Yaskawa INFORM job: KRIS7.JBI

/JOB
//NAME KRIS7
//POS
///NPOS 337,337,337,19,0,0
///TOOL 0
///POSTYPE PULSE
///PULSE
C00000=36471,-76527,-106813,-19264,71481,-77238
C00001=36471,-76527,-106813,-19264,71481,-77238
C00002=63812,-119516,-80644,27282,71106,-59809
C00003=86670,-29465,-24103,33182,93398,-46515
C00004=88663,-31189,-25266,33292,92471,-45985
C00005=89600,-31952,-25776,33339,92036,-45737
C00006=88663,-31189,-25266,33292,92471,-45985
C00007=88663,-31929,-28188,33361,93666,-45629
C00008=101397,-33118,-34088,22474,91022,-41668
C00009=101397,-32934,-33069,22469,90527,-41762
C00010=101397,-33275,-35023,22483,91481,-41581
C00011=104499,20623,14787,23283,115207,-62973
C00012=104352,17765,12486,23220,115200,-63034
C00013=104529,15851,10717,23303,115245,-62949
C00014=104352,17765,12486,23220,115200,-63034
C00015=100086,19810,13187,22516,115799,-63398
C00016=93288,781,-1160,33549,91987,-44264
C00017=95103,1586,-482,33591,91265,-43744
C00018=95638,1156,-842,33600,91054,-43591
C00019=95103,1586,-482,33591,91265,-43744
C00020=100253,-3614,-11898,25466,91372,-41970
C00021=107199,-8537,-17665,19004,89460,-40114
C00022=108350,-8919,-17473,17740,88760,-39873
C00023=102096,-5783,-13006,25389,90415,-41488
C00024=93175,-13453,-24658,25770,96080,-43586
C00025=29596,-126908,-80456,16683,91164,-67663
C00026=130966,-130992,-81417,-14801,93022,34731
C00027=139735,-123676,-71676,-23223,79574,40827
C00028=138444,-123929,-71735,-23429,79144,40460
C00029=134984,-124514,-71869,-23951,78010,39473
C00030=136755,-124231,-71804,-23689,78586,39979
C00031=136306,-124758,-74432,-23664,79703,39597
C00032=105195,-127447,-79852,-15126,73259,28242
C00033=104798,-126140,-77647,-15190,72530,28198
C00034=108375,-128078,-79564,-15067,73342,29336
C00035=112121,-93277,-65445,-16297,96104,47809
C00036=116095,-84503,-58814,-18813,102506,48434
C00037=114391,-86924,-59797,-19239,101506,47972
C00038=116095,-84503,-58814,-18813,102506,48434
C00039=117812,-129995,-81150,-14641,74986,32390
C00040=118791,-92886,-67151,-14205,85296,31516
C00041=116748,-92781,-67110,-14299,84968,30842
C00042=115499,-92681,-67072,-14351,84774,30431
C00043=116748,-92781,-67110,-14299,84968,30842
C00044=116748,-94243,-70296,-14285,86141,30707
C00045=102870,-92009,-70676,-9222,86435,25689
C00046=102870,-90997,-68303,-9229,85506,25758
C00047=102870,-92009,-70676,-9222,86435,25689
C00048=124106,-98193,-79828,-8318,91183,32632
C00049=120990,-117719,-86799,-1028,78019,-83969
C00050=103618,-122878,-84450,-6731,45671,-69045
C00051=107839,-39273,-43881,-11021,86771,-60654
C00052=104365,-32496,-38210,-6982,87775,-60806
C00053=106442,-32422,-37791,-10039,91664,-60187
C00054=103260,-36857,-40680,-8847,97536,-61636
C00055=110992,-39766,-43585,-17340,97602,-59383
C00056=111851,-103912,-94699,-10334,87868,-68255
C00057=100525,-93554,-87313,-9422,87254,-72087
C00058=95765,-72558,-76889,-7644,100510,-59309
C00059=95463,-76426,-71939,-16938,115118,-61391
C00060=97889,-71418,-68275,-18856,117864,-61016
C00061=108072,-63754,-61449,-27079,123073,-58329
C00062=126453,-110744,-88068,-25157,96958,-85114
C00063=124515,-113648,-86106,-25282,93913,-85187
C00064=121942,-111698,-85261,-25663,93564,-86071
C00065=117176,-108078,-83892,-26284,92993,-87738
C00066=122754,-106725,-87203,-25770,97209,-86568
C00067=142865,-91008,-85242,-17891,113758,-73123
C00068=142005,-90205,-84914,-18160,113770,-73464
C00069=93871,-48257,-54590,14207,101968,48555
C00070=106716,17042,-5346,15024,102835,53222
C00071=114740,-14345,-34597,13608,101053,59815
C00072=127078,-3386,-21930,8482,103399,53955
C00073=129218,-1885,-18027,7623,102641,53139
C00074=128838,-13728,-23209,15330,113259,56406
C00075=127376,-6452,-15191,17883,117233,55977
C00076=122058,-3228,-13278,23261,119236,52777
C00077=102997,28917,14853,20600,116287,84527
C00078=102837,-6052,-12869,23266,105489,87265
C00079=105472,-3409,-10021,23525,105335,88236
C00080=105487,-912,-7016,26090,105184,88300
C00081=104416,1445,-8009,23523,106791,88129
C00082=100743,5943,-9423,11985,113108,51981
C00083=104100,-22795,-28366,25068,61310,50210
C00084=122112,-33809,-21710,17217,45375,58941
C00085=131285,-32631,-21327,509,47900,55790
C00086=127059,-25073,-15738,7623,47605,53752
C00087=124156,-6831,-1542,11317,48078,52428
C00088=117469,-7945,-6130,22808,51414,49873
C00089=27812,-119319,-87277,42007,83182,24370
C00090=5621,-139291,-109992,39952,96377,-80222
C00091=5621,-139291,-109992,39952,96377,-80222
C00092=2821,-156918,-126127,-8650,50468,-54614
C00093=2821,-156918,-126127,-8650,75949,-54614
C00094=-114520,-110749,-78127,-8650,75949,-54614
C00095=-130701,-93848,-55732,21077,70446,-8081
C00096=-119736,-94913,-51299,8905,54174,-4125
C00097=-119736,-93106,-48364,9003,53306,-4201
C00098=-119736,-91977,-46540,9068,52768,-4251
C00099=-119736,-92203,-46902,9053,52876,-4241
C00100=-119787,-88445,-45584,8939,53987,-4163
C00101=-119736,-93071,-48307,9005,53289,-4204
C00102=-119736,-93071,-48307,9005,53289,-4204
C00103=-119736,-93071,-48307,9005,53289,-4204
C00104=-119736,-92181,-46869,9053,52867,-4244
C00105=-119736,-92317,-47089,9045,52931,-4239
C00106=-119771,-89498,-46107,8960,53770,-4179
C00107=-119736,-93267,-48625,8993,53383,-4198
C00108=-119736,-93267,-48625,8993,53383,-4198
C00109=-119736,-93267,-48625,8993,53383,-4198
C00110=-119736,-92320,-47093,9047,52931,-4240
C00111=-119736,-92484,-47359,9038,53009,-4233
C00112=-119776,-89491,-46317,8947,53899,-4170
C00113=-119736,-93550,-49086,8979,53518,-4188
C00114=-119736,-95350,-52013,8882,54384,-4113
C00115=-114361,-95392,-52404,-9141,55279,249
C00116=-114361,-93732,-49694,-9231,54474,321
C00117=-114361,-92426,-47572,-9302,53848,379
C00118=-114361,-92561,-47791,-9294,53912,373
C00119=-114623,-89431,-46697,-9121,54806,189
C00120=-114361,-93574,-49437,-9237,54399,330
C00121=-157280,-84649,-46195,2979,55353,-16615
C00122=-157280,-84384,-45724,2984,55199,-16619
C00123=-157280,-83620,-44370,2999,54759,-16630
C00124=-157280,-83726,-44557,2996,54820,-16629
C00125=-155888,-80713,-43363,2571,55586,-16063
C00126=-157843,-85963,-46912,3146,55137,-16842
C00127=-186482,-48100,-18697,2331,50903,-27233
C00128=-187472,-46614,-16803,2745,50531,-27658
C00129=-187472,-45763,-15021,2772,49872,-27676
C00130=-187472,-45864,-15234,2769,49950,-27673
C00131=-185259,-43079,-13610,1852,50319,-26729
C00132=-186728,-50494,-20137,2443,50566,-27343
C00133=-173177,-79635,-34784,14301,47494,-39802
C00134=-170114,-73061,-28660,13270,46626,-38584
C00135=-119904,-88221,-34141,-8998,40682,-15980
C00136=-119767,-102866,-45459,-9162,40143,-15856
C00137=-114881,-103501,-45094,-2719,38974,-10407
C00138=-106437,-88415,-33714,-6684,40170,-6473
C00139=-59844,-64383,-24187,-21266,54434,11788
C00140=-55872,-59424,-21793,-21840,56429,13005
C00141=-56728,-59811,-20829,-16196,48671,13044
C00142=-60192,-86606,-39094,-15561,45595,12032
C00143=-156319,-84382,-37772,-22252,46282,-6119
C00144=-155863,-75602,-29197,-22688,45688,-5754
C00145=-171147,-77982,-28397,2458,37476,-29192
C00146=-189524,-53452,-17206,6300,43588,-32690
C00147=-192814,-47813,-14131,7829,44864,-34109
C00148=-192943,-40170,-9756,2318,45440,-29171
C00149=-168938,-74165,-32389,-22140,45247,-8707
C00150=-139665,-98627,-47692,-8234,50597,-7190
C00151=-157202,-83214,-35232,9186,49733,-29053
C00152=-99055,-87999,-36568,-9269,48061,-5453
C00153=-70072,-109159,-59979,-19142,60032,12699
C00154=-153403,-114623,-61310,-4271,48117,-12926
C00155=-150942,-88287,-33092,-1923,37824,-12225
C00156=-192456,-54522,-18938,15787,50129,-30195
C00157=-191005,-51820,-17697,10248,48517,-24206
C00158=-191538,-49735,-14965,7448,44104,-24349
C00159=-196130,-40875,-10027,9488,46067,-26268
C00160=-193358,-74104,-32741,8607,42709,-25326
C00161=-183204,-85382,-41090,22318,63247,-34683
C00162=-169612,-75107,-30908,21185,58925,-30299
C00163=-165096,-78115,-32117,20755,57090,-28885
C00164=-103759,-88277,-35558,4643,44290,-5139
C00165=-64684,-68765,-27814,-9350,50752,11304
C00166=-59734,-63411,-25340,-10717,52547,13159
C00167=-53928,-55634,-21454,-12166,54909,15247
C00168=-72635,-96956,-47079,-7004,47380,8249
C00169=2821,-156918,-126127,-8650,75949,-54614
C00170=2821,-156918,-126127,-8650,50468,-54614
C00171=5621,-139291,-109992,39952,96377,-80222
C00172=5621,-139291,-109992,39952,96377,-80222
C00173=5621,-139291,-109992,39952,96377,-80222
C00174=5621,-139291,-109992,39952,96377,-80222
C00175=2821,-156918,-126127,-8650,50468,-54614
C00176=2821,-156918,-126127,-8650,75949,-54614
C00177=-103466,-143035,-89833,-18127,44217,664
C00178=-153034,-42791,-3789,574,51224,-21077
C00179=-154411,-23786,22188,-6392,45845,-11810
C00180=-163692,-14831,30793,-3045,43978,-15753
C00181=-162658,-12144,32796,-3380,44162,-15317
C00182=-162658,-10372,35929,-3443,43146,-15280
C00183=-162658,-10822,35136,-3427,43403,-15291
C00184=-163644,-13399,33193,-3102,43239,-15709
C00185=-163644,-12612,34572,-3127,42795,-15690
C00186=-163043,-11060,35746,-3327,42891,-15434
C00187=-163515,-12286,34819,-3170,42815,-15635
C00188=-166152,-32133,5550,-1997,50546,-16952
C00189=-100006,-46830,-3879,-17345,57754,8477
C00190=-55652,-4276,24712,-7053,56203,22524
C00191=-58398,37345,76759,-13956,42466,23962
C00192=-66063,-5406,39790,-11450,41903,20618
C00193=-66063,-3286,43507,-11723,40729,20781
C00194=-66063,-4032,42206,-11625,41137,20723
C00195=-64962,-6235,40444,-12035,41233,21210
C00196=-64962,-5161,42315,-12179,40646,21295
C00197=-65448,-4202,43083,-11996,40600,21078
C00198=-65121,-4851,42561,-12118,40631,21223
C00199=-65121,-17453,19695,-10602,48085,20268
C00200=-72607,-39142,3670,-8250,46011,17274
C00201=-104110,-83683,-24495,4068,39615,3407
C00202=-151806,-110432,-47458,34093,62536,-28079
C00203=-114089,-66317,-11235,33609,49333,-16712
C00204=-80530,-20506,23368,24271,40665,-3524
C00205=-74745,-11317,36142,23442,36289,-1903
C00206=-74745,-9368,39521,24041,35298,-2233
C00207=-85567,-6911,52266,59999,33710,-18160
C00208=-84359,-5993,52985,59939,33118,-17833
C00209=-75543,-10512,38192,25890,35469,-3179
C00210=-78021,-4049,43264,26836,36333,-4217
C00211=-78021,-4049,43264,26836,36333,-4217
C00212=-78560,-2493,44527,27046,36504,-4446
C00213=-78021,-4049,43264,26836,36333,-4217
C00214=-84671,-29838,2091,23749,49176,-3555
C00215=-92002,99,24477,25497,52744,-5935
C00216=-90066,7053,36780,26343,48553,-6224
C00217=-86465,14687,47675,26361,44982,-5590
C00218=-86465,16658,51362,26930,43852,-5949
C00219=-92154,15823,55176,43758,42694,-12452
C00220=-91010,16935,56226,43590,42132,-12113
C00221=-87466,14565,48542,29200,44405,-6685
C00222=-88476,20167,53834,29701,44402,-7193
C00223=-88765,21892,55502,29860,44374,-7348
C00224=-89073,23808,57378,30039,44325,-7522
C00225=-88765,21892,55502,29860,44374,-7348
C00226=-92823,2508,20138,26462,56153,-5606
C00227=-93465,20990,41911,27889,52866,-6816
C00228=-91045,28828,52484,28118,49890,-6598
C00229=-91045,30451,55705,28580,48873,-6919
C00230=-95613,30623,60677,42443,47375,-11939
C00231=-94901,31380,61454,42363,46989,-11750
C00232=-91803,28745,53220,30282,49450,-7369
C00233=-95909,-7710,13963,29350,55596,-7301
C00234=-94576,-67258,-23025,-57506,77870,531
C00235=-146401,-54758,-1647,-68188,44391,-5039
C00236=-142614,-8623,29205,-63903,48682,-7044
C00237=-144464,20682,60858,-67736,45663,-4895
C00238=-144464,22107,63347,-68464,45346,-4423
C00239=-144027,21529,62623,-69515,45942,-4175
C00240=-144859,22233,63313,-69675,45420,-4267
C00241=-144060,21537,62613,-69510,45926,-4186
C00242=-141431,-828,33685,-64125,50152,-7263
C00243=-141985,-10259,26135,-64166,52154,-6525
C00244=-141985,6399,55921,-71703,48228,-1192
C00245=-146205,13772,66109,-74932,44993,-221
C00246=-146205,16430,70459,-76214,44629,596
C00247=-146205,13772,66109,-74932,44993,-221
C00248=-147267,14605,66894,-75256,44365,-306
C00249=-146205,13772,66109,-74932,44993,-221
C00250=-145528,19198,71305,-75151,45267,107
C00251=-145166,21952,74026,-75304,45401,306
C00252=-144772,25167,77279,-75529,45528,563
C00253=-145166,21952,74026,-75304,45401,306
C00254=-145571,-16681,30939,-69324,47370,-3717
C00255=-149532,-31410,21037,-71230,44475,-3428
C00256=-151069,-17310,48414,-81811,41046,2644
C00257=-155207,-6338,62509,-87203,38392,4585
C00258=-155206,-3775,66483,-88647,38310,5410
C00259=-155207,-6338,62509,-87203,38392,4585
C00260=-156672,-5360,63276,-87839,37607,4518
C00261=-155207,-6338,62509,-87203,38392,4585
C00262=-153924,-2552,65524,-86505,39089,4564
C00263=-153389,-833,66935,-86244,39378,4573
C00264=-152779,1247,68674,-85973,39703,4598
C00265=-153389,-833,66935,-86244,39378,4573
C00266=-127211,-52277,-10135,-62715,61377,-4297
C00267=-127211,-63632,-31775,-59501,65152,-7618
C00268=-137468,-45448,-13164,-23993,62707,-9546
C00269=-142031,-34381,-3630,-18745,59946,-9254
C00270=-153480,-23481,18954,-7895,48240,-10284
C00271=-154837,-15674,32352,-7510,43874,-10435
C00272=-154881,-15642,32376,-7496,43872,-10454
C00273=-163905,-10778,37737,-6230,39530,-12164
C00274=-163679,-4139,45223,-21101,38086,-2029
C00275=-164728,-2193,48881,-26376,35092,-528
C00276=-146970,-27557,19782,-29282,44621,5055
C00277=-77984,-28544,12598,-9594,52255,4511
C00278=-87329,-14910,33502,8192,43267,-2149
C00279=-87274,-14870,33531,8174,43265,-2126
C00280=-77526,-7325,39164,4963,42972,2054
C00281=-74703,-2158,47540,17953,35749,-596
C00282=-74957,-595,50445,22566,33903,-2166
C00283=-84696,-19604,28451,27180,39406,-6073
C00284=-87454,-109874,-47340,27972,40441,-7116
C00285=-87454,-109874,-47340,27972,40441,-7116
C00286=-82765,-14870,18327,18756,64283,-30139
C00287=-70453,-8973,33300,17854,53830,-23621
C00288=-79133,18874,57440,18465,54102,-25119
C00289=-78473,16959,55330,17021,52555,-21596
C00290=-81801,-8338,17757,15293,62207,-20035
C00291=-80465,5283,36828,18721,53635,-17767
C00292=-81257,8258,39312,19057,54012,-18385
C00293=-86289,31654,62323,20130,49904,-23761
C00294=-86244,31688,62797,19436,47278,-24020
C00295=-89829,15295,36039,20471,54300,-28399
C00296=-88516,27412,50085,20716,51710,-28378
C00297=-88101,27329,53482,18902,40394,-29830
C00298=-85023,22588,57884,12283,20397,-30375
C00299=-84309,12450,52732,13133,12354,-31131
C00300=-84341,-54767,463,16268,10060,-32559
C00301=-89075,-25175,21935,52893,15017,-40843
C00302=-80632,-262,47578,28811,6370,-27546
C00303=-80188,4143,51700,27800,5999,-27018
C00304=-78793,13633,71285,-46780,-2668,6342
C00305=-83238,-13210,39391,48775,6583,-36846
///LIMIT ON
C00306=-68361,-31604,26984,-58103,4691,13513
///LIMIT OFF
C00307=-66564,-14119,49098,-114271,5370,38931
C00308=-64215,-1164,72142,-148990,11349,55050
///LIMIT ON
C00309=-70339,-38157,28491,-125542,3279,43165
///LIMIT OFF
C00310=-80839,-71335,-37546,-3712,65478,-21646
C00311=-155891,-91755,-42787,-14200,56541,28985
C00312=-171260,-20220,18318,-13706,55116,27713
C00313=-175592,-12005,31520,-10745,48833,21454
C00314=-167202,11927,51151,-10059,48724,20347
C00315=-164608,7730,50211,-16502,43624,19417
C00316=-166381,-4712,22713,-7153,56786,16501
C00317=-164906,4240,35250,-11113,52340,17926
C00318=-163520,9172,39392,-11480,52509,18470
C00319=-157524,37432,66627,-13367,51178,21072
C00320=-157651,33997,63941,-13772,48810,17620
C00321=-157953,21876,39059,-9901,58764,16683
C00322=-154411,30422,52036,-17366,53831,19464
C00323=-154093,33138,54821,-17521,53595,19641
C00324=-155920,26750,56620,-12911,32167,21130
C00325=-156729,27540,61020,-9631,24538,20676
C00326=-159295,5897,40777,-3469,23124,17976
C00327=-161800,-2337,33413,-1605,23382,16874
C00328=-162218,5196,42221,-1134,21829,16584
C00329=-163744,11950,58915,1437,15023,15129
C00330=-178555,-20714,28140,24908,19354,1618
C00331=-170517,-15099,37122,-3989,15402,13548
C00332=-166794,-3567,48220,-19541,26132,18647
C00333=-176772,-46405,12054,26858,15885,1020
C00334=-187852,-124872,-80037,-26712,55091,17871
C00335=-130728,-161100,-136081,-16173,33339,28558
C00336=-1271,-161100,-136081,-16173,33339,28558
BC00000=295309,515546,1075134
BC00001=295309,515546,1075134
BC00002=396955,458142,797628
BC00003=396955,458142,797628
BC00004=396955,458142,797628
BC00005=396955,458142,797628
BC00006=396955,458142,797628
BC00007=396955,458142,797628
BC00008=396955,458142,797628
BC00009=396955,458142,797628
BC00010=396955,458142,797628
BC00011=396955,458142,797628
BC00012=396955,458142,797628
BC00013=396955,458142,797628
BC00014=396955,458142,797628
BC00015=396955,458142,797628
BC00016=396955,458142,797628
BC00017=396955,458142,797628
BC00018=396955,458142,797628
BC00019=396955,458142,797628
BC00020=396955,458142,797628
BC00021=396955,458142,797628
BC00022=396955,458142,797628
BC00023=396955,458142,797628
BC00024=396955,458142,797628
BC00025=396955,458142,797628
BC00026=1315,458142,797628
BC00027=1315,355292,797628
BC00028=1315,355292,797628
BC00029=1315,355292,797628
BC00030=1315,355292,797628
BC00031=1315,355292,797628
BC00032=1315,355292,797628
BC00033=1315,355292,797628
BC00034=1315,355292,797628
BC00035=1315,355292,797628
BC00036=1315,355292,797628
BC00037=1315,355292,797628
BC00038=1315,355292,797628
BC00039=1315,355292,797628
BC00040=1315,355292,797628
BC00041=1315,355292,797628
BC00042=1315,355292,797628
BC00043=1315,355292,797628
BC00044=1315,355292,797628
BC00045=1315,355292,797628
BC00046=1315,355292,797628
BC00047=1315,355292,797628
BC00048=1315,355292,797628
BC00049=1056,429044,516729
BC00050=1056,362244,516729
BC00051=1055,360438,517007
BC00052=786,360252,517036
BC00053=1003,360221,517041
BC00054=1055,360214,517042
BC00055=1055,360214,517042
BC00056=752,360214,695044
BC00057=752,360214,695044
BC00058=752,360214,695044
BC00059=752,360214,695044
BC00060=752,360214,695044
BC00061=752,360214,695044
BC00062=752,360214,695044
BC00063=752,360214,695044
BC00064=752,360214,695044
BC00065=752,360214,695044
BC00066=752,360214,695044
BC00067=752,360214,695044
BC00068=752,503342,695044
BC00069=396955,508258,797628
BC00070=396955,458142,797628
BC00071=396955,458142,797628
BC00072=396955,458142,797628
BC00073=396955,458142,797628
BC00074=396955,458142,797628
BC00075=396955,458142,797628
BC00076=396955,458142,797628
BC00077=396955,458142,797628
BC00078=396955,458142,797628
BC00079=396955,458142,797628
BC00080=396955,458142,797628
BC00081=396955,458142,797628
BC00082=396955,458142,797628
BC00083=396955,458142,516729
BC00084=396955,458142,516729
BC00085=396955,458142,516729
BC00086=396956,458130,516729
BC00087=396955,458142,516729
BC00088=396955,458142,516729
BC00089=396955,458142,516729
BC00090=188270,458142,1013387
BC00091=188270,415623,1052769
BC00092=159481,115072,1070630
BC00093=159481,2193,1070630
BC00094=222221,2193,888573
BC00095=343723,4817,818861
BC00096=343723,4817,818861
BC00097=343723,4817,818861
BC00098=343723,4817,818861
BC00099=343723,4817,818861
BC00100=343723,4817,818861
BC00101=343723,4817,818861
BC00102=285503,4817,818861
BC00103=285503,5201,817244
BC00104=285503,5201,817244
BC00105=285503,5201,817244
BC00106=285503,5201,817244
BC00107=285503,5201,817244
BC00108=225351,5201,824692
BC00109=225351,5201,816215
BC00110=225351,5201,816215
BC00111=225351,5201,816215
BC00112=225351,5201,816215
BC00113=225351,5201,816215
BC00114=225351,5201,816215
BC00115=193660,5201,816215
BC00116=193660,5201,816215
BC00117=193660,5201,816215
BC00118=193660,5201,816215
BC00119=193660,5201,816215
BC00120=193660,5201,816215
BC00121=193660,5201,816215
BC00122=193660,5201,816215
BC00123=193660,5201,816215
BC00124=193660,5201,816215
BC00125=193660,5201,816215
BC00126=193660,5201,816215
BC00127=207415,5201,867665
BC00128=207415,5201,867665
BC00129=207415,5201,867665
BC00130=207415,5201,867665
BC00131=207415,5201,867665
BC00132=207415,5201,867665
BC00133=207415,5201,867665
BC00134=207415,5201,867665
BC00135=207415,5201,867665
BC00136=207415,5201,867665
BC00137=273654,5201,867665
BC00138=273654,5201,867665
BC00139=273654,5201,867665
BC00140=273654,5201,867665
BC00141=273654,5201,867665
BC00142=273654,5201,867665
BC00143=273654,5201,867665
BC00144=225140,12373,867665
BC00145=225140,12373,867665
BC00146=206995,12373,867665
BC00147=206995,12373,867665
BC00148=206995,12373,867665
BC00149=206995,12373,867665
BC00150=268142,12373,867665
BC00151=268142,12373,867665
BC00152=268142,12373,867665
BC00153=268142,12373,867665
BC00154=254581,12373,867665
BC00155=254581,12373,867665
BC00156=254581,12373,867665
BC00157=206517,12373,867665
BC00158=206517,12373,867665
BC00159=206517,12373,867665
BC00160=206517,12373,867665
BC00161=267255,12373,867665
BC00162=267255,12373,867665
BC00163=267255,12373,867665
BC00164=267255,12373,867665
BC00165=267255,12373,867665
BC00166=267255,12373,867665
BC00167=267255,12373,867665
BC00168=267255,12373,867665
BC00169=159481,2193,1070630
BC00170=159481,115072,1070630
BC00171=188270,458142,1013387
BC00172=188270,529869,1013387
BC00173=188270,458142,1013387
BC00174=188270,415623,1052769
BC00175=159481,115072,1070630
BC00176=159481,2193,1070630
BC00177=256379,66753,1051189
BC00178=187914,126248,1051189
BC00179=187914,126248,1051189
BC00180=187915,126247,1051163
BC00181=187915,126247,1051163
BC00182=187915,126247,1051163
BC00183=187915,126247,1051163
BC00184=187915,126247,1051163
BC00185=187915,126247,1051163
BC00186=187915,126247,1051163
BC00187=187915,126247,1051163
BC00188=187915,126247,1051163
BC00189=237533,126248,1051189
BC00190=187914,126248,1051189
BC00191=187914,99975,1051189
BC00192=235697,126248,1051189
BC00193=235697,126248,1051189
BC00194=235697,126248,1051189
BC00195=235697,126248,1051189
BC00196=235697,126248,1051189
BC00197=235697,126248,1051189
BC00198=235697,126248,1051189
BC00199=235697,126248,1051189
BC00200=235697,126248,1051189
BC00201=235697,126248,1051189
BC00202=291851,64960,1051189
BC00203=291851,64960,1051189
BC00204=244068,34238,1051189
BC00205=244068,34238,1051189
BC00206=244068,34238,1051189
BC00207=244068,34238,1051189
BC00208=244068,34238,1051189
BC00209=244068,34238,1051189
BC00210=244068,34238,1051189
BC00211=244068,34238,1051189
BC00212=244068,34238,1051189
BC00213=244068,34238,1051189
BC00214=244068,34238,1051189
BC00215=244068,34238,1051189
BC00216=244068,34238,1051189
BC00217=244068,34238,1051189
BC00218=244068,34238,1051189
BC00219=244068,34238,1051189
BC00220=244068,34238,1051189
BC00221=244068,34238,1051189
BC00222=244068,34238,1051189
BC00223=244068,34238,1051189
BC00224=244068,34238,1051189
BC00225=244068,34238,1051189
BC00226=244068,34238,1051189
BC00227=244068,34238,1051189
BC00228=244067,34238,1051186
BC00229=244067,34238,1051186
BC00230=244067,34238,1051186
BC00231=244067,34238,1051186
BC00232=244067,34238,1051186
BC00233=244067,34238,1051186
BC00234=244067,64961,1051183
BC00235=198013,64961,1051183
BC00236=198013,64961,1051183
BC00237=198013,47917,1051183
BC00238=198013,47917,1051183
BC00239=198013,47917,1051183
BC00240=198013,47917,1051183
BC00241=198013,47917,1051183
BC00242=198013,47917,1051183
BC00243=198013,47917,1051183
BC00244=198013,47917,1051183
BC00245=198013,47917,1051183
BC00246=198013,47917,1051183
BC00247=198013,47917,1051183
BC00248=198013,47917,1051183
BC00249=198013,47917,1051183
BC00250=198013,47917,1051183
BC00251=198013,47917,1051183
BC00252=198013,47917,1051183
BC00253=198013,47917,1051183
BC00254=198013,47917,1051183
BC00255=198013,47917,1051183
BC00256=198013,47917,1051183
BC00257=198013,47917,1051183
BC00258=198013,47917,1051183
BC00259=198013,47917,1051183
BC00260=198013,47917,1051183
BC00261=198013,47917,1051183
BC00262=198013,47917,1051183
BC00263=198013,47917,1051183
BC00264=198013,47917,1051183
BC00265=198013,47917,1051183
BC00266=198013,47917,1051183
BC00267=198013,47917,1051183
BC00268=180161,98336,1051187
BC00269=182927,108294,1051188
BC00270=187693,125451,1051189
BC00271=187914,126248,1051189
BC00272=187914,126248,1051189
BC00273=187914,126248,1051189
BC00274=187914,126248,1051189
BC00275=187914,126248,1051189
BC00276=187914,126248,1051189
BC00277=244068,126248,1051189
BC00278=244068,126248,1051189
BC00279=244068,126248,1051189
BC00280=244068,126248,1051189
BC00281=244068,126248,1051189
BC00282=244068,126248,1051189
BC00283=244068,126248,1051189
BC00284=244068,126248,1051189
BC00285=244068,64960,1051189
BC00286=244068,34238,1051189
BC00287=244068,34238,1051189
BC00288=244068,34238,1051189
BC00289=244068,34238,1051189
BC00290=244068,34238,1051189
BC00291=244068,34238,1051189
BC00292=244068,34238,1051189
BC00293=244068,34238,1051189
BC00294=244068,34238,1051189
BC00295=244068,34238,1051189
BC00296=244068,34238,1051189
BC00297=244068,34238,1051189
BC00298=244068,34238,1051189
BC00299=244068,34238,1051189
BC00300=244068,64960,1051189
BC00301=244068,34238,1051189
BC00302=244068,34238,1051189
BC00303=244068,34238,1051186
BC00304=244068,34238,1051189
BC00305=244068,34238,1051189
BC00306=244068,34238,1051189
BC00307=244067,34238,1051187
BC00308=244068,34238,1051189
BC00309=244068,34238,1051189
BC00310=244068,34238,1051189
BC00311=193074,64960,1051189
BC00312=193074,32459,1055846
BC00313=193074,32459,1055846
BC00314=193074,32459,1055846
BC00315=193075,32459,1055844
BC00316=193074,32459,1055846
BC00317=193074,32459,1055846
BC00318=193074,32459,1055846
BC00319=193074,32459,1055846
BC00320=193074,32459,1055846
BC00321=193074,32459,1055846
BC00322=193074,32459,1055846
BC00323=193074,32459,1055846
BC00324=193074,32459,1055845
BC00325=193074,32459,1055846
BC00326=193074,32459,1055846
BC00327=193074,32459,1055846
BC00328=193074,32459,1055846
BC00329=193074,32459,1055846
BC00330=211313,32459,1055846
BC00331=193074,32459,1055846
BC00332=193074,32459,1055846
BC00333=193074,32459,1055846
BC00334=292209,32459,1055846
BC00335=189350,71534,1070791
BC00336=189350,455301,1070791
EC00000=0,-183832
EC00001=88685,372644
EC00002=88685,372644
EC00003=88685,372644
EC00004=88685,372644
EC00005=88685,372644
EC00006=88685,372644
EC00007=88685,372644
EC00008=88685,372644
EC00009=88685,372644
EC00010=88685,372644
EC00011=88685,372644
EC00012=88685,372644
EC00013=88685,372644
EC00014=88685,372644
EC00015=88685,372644
EC00016=88685,372644
EC00017=88685,372644
EC00018=88685,372644
EC00019=88685,372644
EC00020=88685,372644
EC00021=88685,372644
EC00022=88685,372644
EC00023=88685,372644
EC00024=88685,372644
EC00025=88685,372644
EC00026=88685,372644
EC00027=88685,372644
EC00028=88685,372644
EC00029=88685,372644
EC00030=88685,372644
EC00031=88685,372644
EC00032=88685,372644
EC00033=88685,372644
EC00034=88685,372644
EC00035=88685,372644
EC00036=88685,372644
EC00037=88685,372644
EC00038=88685,372644
EC00039=88685,372644
EC00040=88685,372644
EC00041=88685,372644
EC00042=88685,372644
EC00043=88685,372644
EC00044=88685,372644
EC00045=88685,372644
EC00046=88685,372644
EC00047=88685,372644
EC00048=88685,372644
EC00049=-264893,372644
EC00050=-264893,372644
EC00051=-264346,372644
EC00052=-264290,372644
EC00053=-264280,372644
EC00054=-264278,372644
EC00055=-264278,372644
EC00056=85879,372644
EC00057=85879,372644
EC00058=85879,372644
EC00059=85879,372644
EC00060=85879,372644
EC00061=85879,372644
EC00062=85879,372644
EC00063=85879,372644
EC00064=85879,372644
EC00065=85879,372644
EC00066=85879,372644
EC00067=85879,372644
EC00068=85879,372644
EC00069=88685,372644
EC00070=88685,372644
EC00071=88685,428210
EC00072=88685,428210
EC00073=88685,428210
EC00074=88685,428210
EC00075=88685,428210
EC00076=88685,428210
EC00077=88685,372644
EC00078=88685,372644
EC00079=88685,372644
EC00080=88685,372644
EC00081=88685,372644
EC00082=88685,372644
EC00083=-264893,372644
EC00084=-264893,421244
EC00085=-264893,421244
EC00086=-264894,421244
EC00087=-264893,421244
EC00088=-264893,421244
EC00089=-264893,372644
EC00090=-264890,372644
EC00091=-264890,372644
EC00092=196570,372645
EC00093=492199,372645
EC00094=492199,372645
EC00095=492199,372645
EC00096=492199,372645
EC00097=492199,372645
EC00098=492199,372645
EC00099=492199,372645
EC00100=492199,372645
EC00101=492199,372645
EC00102=492199,372645
EC00103=492199,372645
EC00104=492199,372645
EC00105=492199,372645
EC00106=492199,372645
EC00107=492199,372645
EC00108=492199,372645
EC00109=492199,372645
EC00110=492199,372645
EC00111=492199,372645
EC00112=492199,372645
EC00113=492199,372645
EC00114=492199,372645
EC00115=492199,372645
EC00116=492199,372645
EC00117=492199,372645
EC00118=492199,372645
EC00119=492199,372645
EC00120=492199,372645
EC00121=492199,372645
EC00122=492199,372645
EC00123=492199,372645
EC00124=492199,372645
EC00125=492199,372645
EC00126=492199,372645
EC00127=492199,372645
EC00128=492199,372645
EC00129=492199,372645
EC00130=492199,372645
EC00131=492199,372645
EC00132=492199,372645
EC00133=492199,372645
EC00134=492199,372645
EC00135=492199,372645
EC00136=492199,372645
EC00137=492199,372645
EC00138=492199,372645
EC00139=492199,372645
EC00140=492199,372645
EC00141=492199,372645
EC00142=492199,372645
EC00143=492199,372645
EC00144=492199,372645
EC00145=492199,372645
EC00146=492199,372645
EC00147=492199,372645
EC00148=492199,372645
EC00149=492199,372645
EC00150=492199,372645
EC00151=492199,372645
EC00152=492199,372645
EC00153=492199,372645
EC00154=492199,372645
EC00155=492199,372645
EC00156=492199,372645
EC00157=492199,372645
EC00158=492199,372645
EC00159=492199,372645
EC00160=492199,372645
EC00161=492199,372645
EC00162=492199,372645
EC00163=492199,372645
EC00164=492199,372645
EC00165=492199,372645
EC00166=492199,372645
EC00167=492199,372645
EC00168=492199,372645
EC00169=492199,372645
EC00170=196570,372645
EC00171=-264890,372644
EC00172=-264890,372644
EC00173=-264890,372644
EC00174=-264890,372644
EC00175=196570,372645
EC00176=492199,372645
EC00177=270405,372645
EC00178=270405,372645
EC00179=270405,372645
EC00180=270402,372646
EC00181=270402,372646
EC00182=270402,372646
EC00183=270402,372646
EC00184=270402,372646
EC00185=270402,372646
EC00186=270402,372646
EC00187=270402,372646
EC00188=270402,372646
EC00189=270405,372645
EC00190=270405,372645
EC00191=270405,372645
EC00192=270405,372645
EC00193=270405,372645
EC00194=270405,372645
EC00195=270405,372645
EC00196=270405,372645
EC00197=270405,372645
EC00198=270405,372645
EC00199=270405,372645
EC00200=270405,372645
EC00201=270405,372645
EC00202=447795,372645
EC00203=447795,372645
EC00204=447795,372645
EC00205=447795,372645
EC00206=447795,372645
EC00207=447795,372645
EC00208=447795,372645
EC00209=447795,372645
EC00210=447795,372645
EC00211=447795,372645
EC00212=447795,372645
EC00213=447795,372645
EC00214=447795,372645
EC00215=447795,372645
EC00216=447795,372645
EC00217=447795,372645
EC00218=447795,372645
EC00219=447795,372645
EC00220=447795,372645
EC00221=447795,372645
EC00222=447795,372645
EC00223=447795,372645
EC00224=447795,372645
EC00225=447795,372645
EC00226=447795,372645
EC00227=447795,372645
EC00228=447793,372645
EC00229=447793,372645
EC00230=447793,372645
EC00231=447793,372645
EC00232=447793,372645
EC00233=447793,372645
EC00234=447791,372645
EC00235=447791,372645
EC00236=447791,372645
EC00237=447791,372645
EC00238=447791,372645
EC00239=447791,372645
EC00240=447791,372645
EC00241=447791,372645
EC00242=447791,372645
EC00243=447791,372645
EC00244=447791,372645
EC00245=447791,372645
EC00246=447791,372645
EC00247=447791,372645
EC00248=447791,372645
EC00249=447791,372645
EC00250=447791,372645
EC00251=447791,372645
EC00252=447791,372645
EC00253=447791,372645
EC00254=447791,372645
EC00255=447791,372645
EC00256=447791,372645
EC00257=447791,372645
EC00258=447791,372645
EC00259=447791,372645
EC00260=447791,372645
EC00261=447791,372645
EC00262=447791,372645
EC00263=447791,372645
EC00264=447791,372645
EC00265=447791,372645
EC00266=447791,372645
EC00267=447791,372645
EC00268=333615,372645
EC00269=311064,372645
EC00270=272209,372645
EC00271=270405,372645
EC00272=270405,372645
EC00273=270405,372645
EC00274=270405,372645
EC00275=270405,372645
EC00276=270405,372645
EC00277=270405,372645
EC00278=270405,372645
EC00279=270405,372645
EC00280=270405,372645
EC00281=270405,372645
EC00282=270405,372645
EC00283=270405,372645
EC00284=270405,372645
EC00285=447795,372645
EC00286=447795,372645
EC00287=447795,372645
EC00288=447795,372645
EC00289=447795,372645
EC00290=447795,372645
EC00291=447795,372645
EC00292=447795,372645
EC00293=447795,372645
EC00294=447795,372645
EC00295=447795,372645
EC00296=447795,372645
EC00297=447795,372645
EC00298=447795,372645
EC00299=447795,372645
EC00300=447795,372645
EC00301=447795,372645
EC00302=447795,372645
EC00303=447794,372645
EC00304=447795,372645
EC00305=447795,372645
EC00306=447795,372645
EC00307=447794,372646
EC00308=447795,372645
EC00309=447795,372645
EC00310=447795,372645
EC00311=447795,372645
EC00312=447795,372645
EC00313=447795,372645
EC00314=447795,372645
EC00315=447794,372645
EC00316=447795,372645
EC00317=447795,372645
EC00318=447795,372645
EC00319=447795,372645
EC00320=447795,372645
EC00321=447795,372645
EC00322=447795,372645
EC00323=447795,372645
EC00324=447794,372646
EC00325=447795,372645
EC00326=447795,372645
EC00327=447795,372645
EC00328=447795,372645
EC00329=447795,372645
EC00330=447795,372645
EC00331=447795,372645
EC00332=447795,372645
EC00333=447795,372645
EC00334=447795,372645
EC00335=71624,372645
EC00336=-15446,372645
///POSTYPE BASE
///RECTAN
///RCONF 0,0,0,0,1,0,0,0,0,0,0,0,0,0,0,0,0,0,0,0,0,0,0,0
P00006=2.006,1.622,-0.565,0.0000,0.0000,0.0000
P00021=0.073,2.058,-0.109,0.0000,0.0000,0.0000
P00022=2.006,1.622,-0.565,0.0000,0.0000,0.0000
///RCONF 0,0,0,0,0,0,0,0,0,0,0,0,0,0,0,0,0,0,0,0,0,0,0,0
P00023=-2.957,-4.083,2.762,0.0000,0.0000,0.0000
P00024=-1.466,-0.226,-0.419,0.0000,0.0000,0.0000
P00025=3.643,0.007,-2.585,0.0000,0.0000,0.0000
P00026=2.644,0.055,-2.583,0.0000,0.0000,0.0000
P00032=-0.423,0.157,3.222,0.0000,0.0000,0.0000
P00033=0.854,-1.099,3.047,0.0000,0.0000,0.0000
///RCONF 0,0,0,0,1,0,0,0,0,0,0,0,0,0,0,0,0,0,0,0,0,0,0,0
P00034=-8.151,9.743,-4.393,0.0000,0.0000,0.0000
///RCONF 0,0,0,0,0,0,0,0,0,0,0,0,0,0,0,0,0,0,0,0,0,0,0,0
P00035=0.390,-0.027,1.040,0.0000,0.0000,0.0000
P00042=-0.220,0.371,-0.613,0.0000,0.0000,0.0000
P00043=-0.179,-5.890,-3.227,0.0000,0.0000,0.0000
P00044=-8.560,-7.557,-5.232,0.0000,0.0000,0.0000
P00045=-8.836,-6.632,-1.438,0.0000,0.0000,0.0000
P00046=-7.725,-0.107,-2.878,0.0000,0.0000,0.0000
P00048=-10.315,0.035,-3.101,0.0000,0.0000,0.0000
P00049=-9.638,1.690,-2.627,0.0000,0.0000,0.0000
P00050=-0.123,2.174,-1.314,0.0000,0.0000,0.0000
//INST
///DATE 2024/12/19 20:24
///ATTR SC,RW
///GROUP1 RB1,BS1
///GROUP2 ST1
NOP
MOVJ C00000 BC00000 VJ=100.00  +MOVJ EC00000 VJ=100.00
MOVJ C00001 BC00001 VJ=100.00  +MOVJ EC00001 VJ=100.00
CALL JOB:CLEAN-R1_KM_NEW
MOVJ C00002 BC00002 VJ=100.00  +MOVJ EC00002 VJ=100.00
MOVJ C00003 BC00003 VJ=50.00  +MOVJ EC00003 VJ=50.00
SMOVL C00004 BC00004 V=83.3  +MOVJ EC00004
SREFP 3 C00005 BC00005  +REFP EC00005
CALL JOB:SEARCH-R1-S13D
SET P032 P006
SFTON3D P032
SMOVL C00006 BC00006 V=60.0  +MOVJ EC00006
SMOVL C00007 BC00007 V=133.3  +MOVJ EC00007
SMOVL C00008 BC00008 V=133.3  +MOVJ EC00008
SREFP 3 C00009 BC00009  +REFP EC00009
CALL JOB:SEARCH-R1-S13D
SET P032 P006
SFTON3D P032
SMOVL C00010 BC00010 V=60.0  +MOVJ EC00010
SMOVL C00011 BC00011 V=133.3  +MOVJ EC00011
SMOVL C00012 BC00012 V=133.3  +MOVJ EC00012
SREFP 3 C00013 BC00013  +REFP EC00013
CALL JOB:SEARCH-R1-S13D
SET P032 P006
SFTON3D P032
SFTOF3D
SMOVL C00014 BC00014 V=133.3  +MOVJ EC00014
SMOVL C00015 BC00015 V=200.0  +MOVJ EC00015
SFTOF3D
'S1
MOVJ C00016 BC00016 VJ=50.00  +MOVJ EC00016 VJ=50.00
'S2
SMOVL C00017 BC00017 V=60.0  +MOVJ EC00017
SREFP 3 C00018 BC00018  +REFP EC00018
CALL JOB:SEARCH-R1-S13D
SET P033 P006
SFTON3D P033
SMOVL C00019 BC00019 V=60.0  +MOVJ EC00019
SMOVL C00020 BC00020 V=133.3  +MOVJ EC00020
SMOVL C00021 BC00021 V=133.3  +MOVJ EC00021
SREFP 3 C00022 BC00022  +REFP EC00022
CALL JOB:SEARCH-R1-S13D
SET P033 P006
SFTON3D P033
SFTOF3D
SMOVL C00023 BC00023 V=83.3  +MOVJ EC00023
MOVJ C00024 BC00024 VJ=60.00  +MOVJ EC00024 VJ=60.00
MOVJ C00025 BC00025 VJ=60.00  +MOVJ EC00025 VJ=60.00
MOVJ C00026 BC00026 VJ=100.00  +MOVJ EC00026 VJ=60.00
MOVJ C00027 BC00027 VJ=60.00  +MOVJ EC00027 VJ=60.00
SMOVL C00028 BC00028 V=60.0  +MOVJ EC00028
SREFP 3 C00029 BC00029  +REFP EC00029
CALL JOB:SEARCH-R1-S13D
SET P034 P006
SFTON3D P034
SMOVL C00030 BC00030 V=60.0  +MOVJ EC00030
SMOVL C00031 BC00031 V=83.3  +MOVJ EC00031
SMOVL C00032 BC00032 V=83.3  +MOVJ EC00032
SREFP 3 C00033 BC00033  +REFP EC00033
CALL JOB:SEARCH-R1-S13D
SET P034 P006
SFTON3D P034
SMOVL C00034 BC00034 V=100.0  +MOVJ EC00034
SMOVL C00035 BC00035 V=133.3  +MOVJ EC00035
SMOVL C00036 BC00036 V=133.3  +MOVJ EC00036
SREFP 3 C00037 BC00037  +REFP EC00037
CALL JOB:SEARCH-R1-S13D
SET P034 P006
SFTON3D P034
SMOVL C00038 BC00038 V=133.3  +MOVJ EC00038
SMOVL C00039 BC00039 V=133.3  +MOVJ EC00039
SMOVL C00040 BC00040 V=250.0  +MOVJ EC00040
SMOVL C00041 BC00041 V=60.0  +MOVJ EC00041
SREFP 3 C00042 BC00042  +REFP EC00042
CALL JOB:SEARCH-R1-S13D
SET P035 P006
SFTON3D P035
SMOVL C00043 BC00043 V=60.0  +MOVJ EC00043
SMOVL C00044 BC00044 V=250.0  +MOVJ EC00044
SMOVL C00045 BC00045 V=250.0  +MOVJ EC00045
SREFP 3 C00046 BC00046  +REFP EC00046
CALL JOB:SEARCH-R1-S13D
SET P035 P006
SFTON3D P035
SMOVL C00047 BC00047 V=166.7  +MOVJ EC00047
SFTOF3D
MOVJ C00048 BC00048 VJ=30.00  +MOVJ EC00048 VJ=15.00
MOVJ C00049 BC00049 VJ=100.00  +MOVJ EC00049 VJ=50.00
MACRO1 MJ#(0) ARGF9
MOVJ C00050 BC00050 VJ=100.00  +MOVJ EC00050 VJ=15.00
SMOVL C00051 BC00051 V=666.7  +MOVJ EC00051
SFTON3D P035
SMOVL C00052 BC00052 V=166.7  +MOVJ EC00052
ARCON
SMOVL C00053 BC00053 V=6.7  +MOVJ EC00053
SMOVL C00054 BC00054 V=6.7  +MOVJ EC00054
ARCOF
TIMER T=1.00
SMOVL C00055 BC00055 V=166.7  +MOVJ EC00055
SFTOF3D
MOVJ C00056 BC00056 VJ=20.00  +MOVJ EC00056 VJ=100.00
MOVJ C00057 BC00057 VJ=15.00  +MOVJ EC00057 VJ=100.00
SFTON3D P035
SMOVL C00058 BC00058 V=166.7  +MOVJ EC00058
ARCON
SFTON3D P034
SMOVL C00059 BC00059 V=8.3  +MOVJ EC00059
SMOVL C00060 BC00060 V=8.3  +MOVJ EC00060
ARCOF
SMOVL C00061 BC00061 V=166.7  +MOVJ EC00061
SMOVL C00062 BC00062 V=500.0  +MOVJ EC00062
SMOVL C00063 BC00063 V=166.7  +MOVJ EC00063
ARCON
SMOVL C00064 BC00064 V=7.5  +MOVJ EC00064
SMOVL C00065 BC00065 V=7.5  +MOVJ EC00065
ARCOF
SFTOF3D
MOVJ C00066 BC00066 VJ=30.00  +MOVJ EC00066 VJ=60.00
MOVJ C00067 BC00067 VJ=100.00  +MOVJ EC00067 VJ=50.00
MOVJ C00068 BC00068 VJ=100.00  +MOVJ EC00068 VJ=15.00
MOVJ C00069 BC00069 VJ=100.00  +MOVJ EC00069 VJ=100.00
MOVJ C00070 BC00070 VJ=50.00  +MOVJ EC00070 VJ=50.00
SFTOF3D
MOVJ C00071 BC00071 VJ=100.00  +MOVJ EC00071 VJ=100.00
MOVJ C00072 BC00072 VJ=100.00  +MOVJ EC00072 VJ=100.00
SFTON3D P033
SMOVL C00073 BC00073 V=166.7  +MOVJ EC00073
ARCON
SFTON3D P032
SMOVL C00074 BC00074 V=8.3  +MOVJ EC00074
SMOVL C00075 BC00075 V=8.3  +MOVJ EC00075
ARCOF
SMOVL C00076 BC00076 V=166.7  +MOVJ EC00076
SMOVL C00077 BC00077 V=666.7  +MOVJ EC00077
SMOVL C00078 BC00078 V=133.3  +MOVJ EC00078
ARCON
SMOVL C00079 BC00079 V=7.5  +MOVJ EC00079
SMOVL C00080 BC00080 V=7.5  +MOVJ EC00080
ARCOF
SFTOF3D
SMOVL C00081 BC00081 V=133.3  +MOVJ EC00081
MOVJ C00082 BC00082 VJ=50.00  +MOVJ EC00082 VJ=50.00
MOVJ C00083 BC00083 VJ=100.00  +MOVJ EC00083 VJ=100.00
MOVJ C00084 BC00084 VJ=100.00  +MOVJ EC00084 VJ=100.00
SFTON3D P033
SMOVL C00085 BC00085 V=133.3  +MOVJ EC00085
ARCON
SMOVL C00086 BC00086 V=7.5  +MOVJ EC00086
ARCON
SMOVL C00087 BC00087 V=7.5  +MOVJ EC00087
ARCOF
MOVJ C00088 BC00088 VJ=50.00  +MOVJ EC00088 VJ=50.00
MOVJ C00089 BC00089 VJ=100.00  +MOVJ EC00089 VJ=100.00
CALL JOB:CLEAN-R1_KM_NEW
PAUSE
PAUSE
PAUSE
'TRZEBA NOWY PROGRAM NA NOZ
MOVJ C00090 BC00090 VJ=100.00  +MOVJ EC00090 VJ=100.00
MOVJ C00091 BC00091 VJ=100.00  +MOVJ EC00091 VJ=100.00
MOVJ C00092 BC00092 VJ=100.00  +MOVJ EC00092 VJ=100.00
MOVJ C00093 BC00093 VJ=100.00  +MOVJ EC00093 VJ=100.00
MOVJ C00094 BC00094 VJ=100.00  +MOVJ EC00094 VJ=100.00
MOVJ C00095 BC00095 VJ=100.00  +MOVJ EC00095 VJ=100.00
MOVL C00096 BC00096 V=250.0  +MOVJ EC00096 VJ=100.00
SMOVL C00097 BC00097 V=100.0  +MOVJ EC00097
SREFP 3 C00098 BC00098  +REFP EC00098
CALL JOB:SEARCH-R1-S13D
SET P021 P006
SFTON3D P021
SMOVL C00099 BC00099 V=100.0  +MOVJ EC00099
SREFP 3 C00100 BC00100  +REFP EC00100
CALL JOB:SEARCH-R1-S13D
SET P021 P006
SFTON3D P021
SMOVL C00101 BC00101 V=100.0  +MOVJ EC00101
SFTOF3D
MOVL C00102 BC00102 V=250.0  +MOVJ EC00102 VJ=100.00
SMOVL C00103 BC00103 V=100.0  +MOVJ EC00103
SREFP 3 C00104 BC00104  +REFP EC00104
CALL JOB:SEARCH-R1-S13D
SET P022 P006
SFTON3D P022
SMOVL C00105 BC00105 V=100.0  +MOVJ EC00105
SREFP 3 C00106 BC00106  +REFP EC00106
CALL JOB:SEARCH-R1-S13D
SET P022 P006
SFTON3D P022
SMOVL C00107 BC00107 V=100.0  +MOVJ EC00107
SFTOF3D
MOVL C00108 BC00108 V=250.0  +MOVJ EC00108 VJ=100.00
SMOVL C00109 BC00109 V=100.0  +MOVJ EC00109
SREFP 3 C00110 BC00110  +REFP EC00110
CALL JOB:SEARCH-R1-S13D
SET P023 P006
SFTON3D P023
SMOVL C00111 BC00111 V=100.0  +MOVJ EC00111
SREFP 3 C00112 BC00112  +REFP EC00112
CALL JOB:SEARCH-R1-S13D
SET P023 P006
SFTON3D P023
SMOVL C00113 BC00113 V=100.0  +MOVJ EC00113
SFTOF3D
MOVL C00114 BC00114 V=250.0  +MOVJ EC00114 VJ=100.00
MOVL C00115 BC00115 V=250.0  +MOVJ EC00115 VJ=100.00
SMOVL C00116 BC00116 V=100.0  +MOVJ EC00116
SREFP 3 C00117 BC00117  +REFP EC00117
CALL JOB:SEARCH-R1-S13D
SET P024 P006
SFTON3D P024
SMOVL C00118 BC00118 V=100.0  +MOVJ EC00118
SREFP 3 C00119 BC00119  +REFP EC00119
CALL JOB:SEARCH-R1-S13D
SET P024 P006
SFTON3D P024
SMOVL C00120 BC00120 V=100.0  +MOVJ EC00120
SFTOF3D
MOVL C00121 BC00121 V=250.0  +MOVJ EC00121 VJ=100.00
SMOVL C00122 BC00122 V=100.0  +MOVJ EC00122
SREFP 3 C00123 BC00123  +REFP EC00123
CALL JOB:SEARCH-R1-S13D
SET P025 P006
SFTON3D P025
SMOVL C00124 BC00124 V=100.0  +MOVJ EC00124
SREFP 3 C00125 BC00125  +REFP EC00125
CALL JOB:SEARCH-R1-S13D
SET P025 P006
SFTON3D P025
SMOVL C00126 BC00126 V=100.0  +MOVJ EC00126
SFTOF3D
MOVL C00127 BC00127 V=250.0  +MOVJ EC00127 VJ=100.00
SMOVL C00128 BC00128 V=100.0  +MOVJ EC00128
SREFP 3 C00129 BC00129  +REFP EC00129
CALL JOB:SEARCH-R1-S13D
SET P026 P006
SFTON3D P026
SMOVL C00130 BC00130 V=100.0  +MOVJ EC00130
SREFP 3 C00131 BC00131  +REFP EC00131
CALL JOB:SEARCH-R1-S13D
SET P026 P006
SFTON3D P026
SMOVL C00132 BC00132 V=166.7  +MOVJ EC00132
SFTOF3D
MOVL C00133 BC00133 V=333.3  +MOVJ EC00133 VJ=100.00
SFTON3D P025
MACRO1 MJ#(0) ARGF9
MOVL C00134 BC00134 V=166.7  +MOVJ EC00134 VJ=100.00
ARCON
SFTON3D P024
MOVL C00135 BC00135 V=10.0  +MOVJ EC00135 VJ=100.00
ARCOF
SFTOF3D
MOVL C00136 BC00136 V=250.0  +MOVJ EC00136 VJ=100.00
MOVL C00137 BC00137 V=250.0  +MOVJ EC00137 VJ=100.00
SFTON3D P022
MOVL C00138 BC00138 V=166.7  +MOVJ EC00138 VJ=100.00
ARCON
SFTON3D P021
MOVL C00139 BC00139 V=10.0  +MOVJ EC00139 VJ=100.00
ARCOF
MOVL C00140 BC00140 V=25.0  +MOVJ EC00140 VJ=100.00
ARCON
MOVL C00141 BC00141 V=10.0  +MOVJ EC00141 VJ=100.00
ARCOF
MOVL C00142 BC00142 V=250.0  +MOVJ EC00142 VJ=100.00
MOVL C00143 BC00143 V=250.0  +MOVJ EC00143 VJ=100.00
MOVL C00144 BC00144 V=250.0  +MOVJ EC00144 VJ=100.00
SFTON3D P025
MOVL C00145 BC00145 V=166.7  +MOVJ EC00145 VJ=100.00
ARCON
SFTON3D P026
MOVL C00146 BC00146 V=10.0  +MOVJ EC00146 VJ=100.00
ARCOF
MOVL C00147 BC00147 V=25.0  +MOVJ EC00147 VJ=100.00
ARCON
MOVL C00148 BC00148 V=10.0  +MOVJ EC00148 VJ=100.00
ARCOF
SFTOF3D
MOVL C00149 BC00149 V=250.0  +MOVJ EC00149 VJ=100.00
MOVL C00150 BC00150 V=250.0  +MOVJ EC00150 VJ=100.00
SFTON3D P023
MOVL C00151 BC00151 V=166.7  +MOVJ EC00151 VJ=100.00
ARCON
SFTON3D P022
MOVL C00152 BC00152 V=10.0  +MOVJ EC00152 VJ=100.00
ARCOF
SFTOF3D
MOVL C00153 BC00153 V=250.0  +MOVJ EC00153 VJ=100.00
MOVL C00154 BC00154 V=250.0  +MOVJ EC00154 VJ=100.00
SFTON3D P024
MOVL C00155 BC00155 V=166.7  +MOVJ EC00155 VJ=100.00
ARCON
SFTON3D P025
MOVL C00156 BC00156 V=11.7  +MOVJ EC00156 VJ=100.00
SFTON3D P026
MOVL C00157 BC00157 V=11.7  +MOVJ EC00157 VJ=100.00
ARCOF
MOVL C00158 BC00158 V=25.0  +MOVJ EC00158 VJ=100.00
ARCON
MOVL C00159 BC00159 V=11.7  +MOVJ EC00159 VJ=100.00
ARCOF
SFTOF3D
MOVL C00160 BC00160 V=250.0  +MOVJ EC00160 VJ=100.00
MOVL C00161 BC00161 V=250.0  +MOVJ EC00161 VJ=100.00
SFTON3D P023
MOVL C00162 BC00162 V=166.7  +MOVJ EC00162 VJ=100.00
ARCON
MOVL C00163 BC00163 V=10.8  +MOVJ EC00163 VJ=100.00
SFTON3D P022
MOVL C00164 BC00164 V=10.8  +MOVJ EC00164 VJ=100.00
SFTON3D P021
MOVL C00165 BC00165 V=10.8  +MOVJ EC00165 VJ=100.00
ARCOF
MOVL C00166 BC00166 V=25.0  +MOVJ EC00166 VJ=100.00
ARCON
MOVL C00167 BC00167 V=10.8  +MOVJ EC00167 VJ=100.00
ARCOF
SFTOF3D
MOVL C00168 BC00168 V=250.0  +MOVJ EC00168 VJ=100.00
MOVJ C00169 BC00169 VJ=100.00  +MOVJ EC00169 VJ=100.00
MOVJ C00170 BC00170 VJ=100.00  +MOVJ EC00170 VJ=100.00
MOVJ C00171 BC00171 VJ=100.00  +MOVJ EC00171 VJ=100.00
MOVJ C00172 BC00172 VJ=100.00  +MOVJ EC00172 VJ=100.00
PAUSE
CALL JOB:CLEAN-R1_KM_NEW
'TRZEBA NOWY PROGRAM NA NOZ
MOVJ C00173 BC00173 VJ=100.00  +MOVJ EC00173 VJ=100.00
MOVJ C00174 BC00174 VJ=100.00  +MOVJ EC00174 VJ=100.00
MOVJ C00175 BC00175 VJ=100.00  +MOVJ EC00175 VJ=100.00
MOVJ C00176 BC00176 VJ=100.00  +MOVJ EC00176 VJ=100.00
MOVJ C00177 BC00177 VJ=100.00  +MOVJ EC00177 VJ=50.00
MOVJ C00178 BC00178 VJ=100.00  +MOVJ EC00178 VJ=50.00
MOVJ C00179 BC00179 VJ=15.00  +MOVJ EC00179 VJ=15.00
MOVJ C00180 BC00180 VJ=15.00  +MOVJ EC00180 VJ=50.00
SMOVL C00181 BC00181 V=83.3  +MOVJ EC00181
SREFP 3 C00182 BC00182  +REFP EC00182
CALL JOB:SEARCH-R1-S13D
SET P042 P006
SFTON3D P042
SMOVL C00183 BC00183 V=60.0  +MOVJ EC00183
SMOVL C00184 BC00184 V=133.3  +MOVJ EC00184
SMOVL C00185 BC00185 V=133.3  +MOVJ EC00185
SREFP 3 C00186 BC00186  +REFP EC00186
CALL JOB:SEARCH-R1-S13D
SET P042 P006
SFTON3D P042
SMOVL C00187 BC00187 V=60.0  +MOVJ EC00187
SFTOF3D
MOVJ C00188 BC00188 VJ=15.00  +MOVJ EC00188 VJ=15.00
MOVJ C00189 BC00189 VJ=15.00  +MOVJ EC00189 VJ=15.00
MOVJ C00190 BC00190 VJ=15.00  +MOVJ EC00190 VJ=15.00
MOVJ C00191 BC00191 VJ=15.00  +MOVJ EC00191 VJ=15.00
SMOVL C00192 BC00192 V=83.3  +MOVJ EC00192
SREFP 3 C00193 BC00193  +REFP EC00193
CALL JOB:SEARCH-R1-S13D
SET P043 P006
SFTON3D P043
SMOVL C00194 BC00194 V=60.0  +MOVJ EC00194
SMOVL C00195 BC00195 V=133.3  +MOVJ EC00195
SMOVL C00196 BC00196 V=133.3  +MOVJ EC00196
SREFP 3 C00197 BC00197  +REFP EC00197
CALL JOB:SEARCH-R1-S13D
SET P043 P006
SFTON3D P043
SMOVL C00198 BC00198 V=60.0  +MOVJ EC00198
MOVJ C00199 BC00199 VJ=30.00  +MOVJ EC00199 VJ=30.00
SFTOF3D
MOVJ C00200 BC00200 VJ=30.00  +MOVJ EC00200 VJ=30.00
MOVJ C00201 BC00201 VJ=30.00  +MOVJ EC00201 VJ=30.00
MOVJ C00202 BC00202 VJ=50.00  +MOVJ EC00202 VJ=50.00
MOVJ C00203 BC00203 VJ=50.00  +MOVJ EC00203 VJ=50.00
SFTOF3D
MOVJ C00204 BC00204 VJ=30.00  +MOVJ EC00204 VJ=30.00
SMOVL C00205 BC00205 V=83.3  +MOVJ EC00205
SREFP 3 C00206 BC00206  +REFP EC00206
CALL JOB:SEARCH-R1-S13D
SET P044 P006
SFTON3D P044
SMOVL C00207 BC00207 V=100.0  +MOVJ EC00207
SREFP 3 C00208 BC00208  +REFP EC00208
CALL JOB:SEARCH-R1-S13D
SET P044 P006
SFTON3D P044
SMOVL C00209 BC00209 V=133.3  +MOVJ EC00209
SMOVL C00210 BC00210 V=250.0  +MOVJ EC00210
SMOVL C00211 BC00211 V=133.3  +MOVJ EC00211
SREFP 3 C00212 BC00212  +REFP EC00212
CALL JOB:SEARCH-R1-S13D
SET P044 P006
SFTON3D P044
SMOVL C00213 BC00213 V=133.3  +MOVJ EC00213
SFTOF3D
MOVJ C00214 BC00214 VJ=30.00  +MOVJ EC00214 VJ=15.00
MOVJ C00215 BC00215 VJ=30.00  +MOVJ EC00215 VJ=15.00
MOVJ C00216 BC00216 VJ=30.00  +MOVJ EC00216 VJ=15.00
SMOVL C00217 BC00217 V=250.0  +MOVJ EC00217
SREFP 3 C00218 BC00218  +REFP EC00218
CALL JOB:SEARCH-R1-S13D
SET P045 P006
SFTON3D P045
SMOVL C00219 BC00219 V=250.0  +MOVJ EC00219
SREFP 3 C00220 BC00220  +REFP EC00220
CALL JOB:SEARCH-R1-S13D
SET P045 P006
SFTON3D P045
SMOVL C00221 BC00221 V=250.0  +MOVJ EC00221
SMOVL C00222 BC00222 V=250.0  +MOVJ EC00222
SMOVL C00223 BC00223 V=166.7  +MOVJ EC00223
SREFP 3 C00224 BC00224  +REFP EC00224
CALL JOB:SEARCH-R1-S13D
SET P045 P006
SFTON3D P045
SMOVL C00225 BC00225 V=250.0  +MOVJ EC00225
SFTOF3D
MOVJ C00226 BC00226 VJ=30.00  +MOVJ EC00226 VJ=15.00
MOVJ C00227 BC00227 VJ=30.00  +MOVJ EC00227 VJ=15.00
SMOVL C00228 BC00228 V=250.0  +MOVJ EC00228
SREFP 3 C00229 BC00229  +REFP EC00229
CALL JOB:SEARCH-R1-S13D
SET P046 P006
SFTON3D P046
SMOVL C00230 BC00230 V=250.0  +MOVJ EC00230
SREFP 3 C00231 BC00231  +REFP EC00231
CALL JOB:SEARCH-R1-S13D
SET P046 P006
SFTON3D P046
SMOVL C00232 BC00232 V=250.0  +MOVJ EC00232
SFTOF3D
MOVJ C00233 BC00233 VJ=30.00  +MOVJ EC00233 VJ=15.00
MOVJ C00234 BC00234 VJ=30.00  +MOVJ EC00234 VJ=15.00
MOVJ C00235 BC00235 VJ=30.00  +MOVJ EC00235 VJ=15.00
MOVJ C00236 BC00236 VJ=30.00  +MOVJ EC00236 VJ=15.00
SMOVL C00237 BC00237 V=250.0  +MOVJ EC00237
SREFP 3 C00238 BC00238  +REFP EC00238
CALL JOB:SEARCH-R1-S13D
SET P048 P006
SFTON3D P048
SMOVL C00239 BC00239 V=250.0  +MOVJ EC00239
SREFP 3 C00240 BC00240  +REFP EC00240
CALL JOB:SEARCH-R1-S13D
SET P048 P006
SFTON3D P048
SMOVL C00241 BC00241 V=250.0  +MOVJ EC00241
MOVJ C00242 BC00242 VJ=30.00  +MOVJ EC00242 VJ=15.00
SFTOF3D
MOVJ C00243 BC00243 VJ=30.00  +MOVJ EC00243 VJ=15.00
MOVJ C00244 BC00244 VJ=30.00  +MOVJ EC00244 VJ=15.00
SMOVL C00245 BC00245 V=166.7  +MOVJ EC00245
SREFP 3 C00246 BC00246  +REFP EC00246
CALL JOB:SEARCH-R1-S13D
SET P049 P006
SFTON3D P049
SMOVL C00247 BC00247 V=166.7  +MOVJ EC00247
SREFP 3 C00248 BC00248  +REFP EC00248
CALL JOB:SEARCH-R1-S13D
SET P049 P006
SFTON3D P049
SMOVL C00249 BC00249 V=166.7  +MOVJ EC00249
SMOVL C00250 BC00250 V=166.7  +MOVJ EC00250
SMOVL C00251 BC00251 V=166.7  +MOVJ EC00251
SREFP 3 C00252 BC00252  +REFP EC00252
CALL JOB:SEARCH-R1-S13D
SET P049 P006
SFTON3D P049
SMOVL C00253 BC00253 V=166.7  +MOVJ EC00253
SFTOF3D
MOVJ C00254 BC00254 VJ=30.00  +MOVJ EC00254 VJ=30.00
MOVJ C00255 BC00255 VJ=30.00  +MOVJ EC00255 VJ=30.00
MOVJ C00256 BC00256 VJ=30.00  +MOVJ EC00256 VJ=15.00
SMOVL C00257 BC00257 V=250.0  +MOVJ EC00257
SREFP 3 C00258 BC00258  +REFP EC00258
CALL JOB:SEARCH-R1-S13D
SET P050 P006
SFTON3D P050
SMOVL C00259 BC00259 V=250.0  +MOVJ EC00259
SREFP 3 C00260 BC00260  +REFP EC00260
CALL JOB:SEARCH-R1-S13D
SET P050 P006
SFTON3D P050
SMOVL C00261 BC00261 V=250.0  +MOVJ EC00261
SMOVL C00262 BC00262 V=250.0  +MOVJ EC00262
SMOVL C00263 BC00263 V=166.7  +MOVJ EC00263
SREFP 3 C00264 BC00264  +REFP EC00264
CALL JOB:SEARCH-R1-S13D
SET P050 P006
SFTON3D P050
SMOVL C00265 BC00265 V=166.7  +MOVJ EC00265
SFTOF3D
MOVJ C00266 BC00266 VJ=30.00  +MOVJ EC00266 VJ=15.00
MOVJ C00267 BC00267 VJ=30.00  +MOVJ EC00267 VJ=15.00
MOVJ C00268 BC00268 VJ=30.00  +MOVJ EC00268 VJ=15.00
MOVJ C00269 BC00269 VJ=30.00  +MOVJ EC00269 VJ=30.00
MOVJ C00270 BC00270 VJ=30.00  +MOVJ EC00270 VJ=30.00
MACRO1 MJ#(0) ARGF9
SFTON3D P042
SMOVL C00271 BC00271 V=166.7  +MOVJ EC00271
ARCON
SMOVC C00272 BC00272 V=8.3  +MOVJ EC00272
SMOVC C00273 BC00273 V=8.3  +MOVJ EC00273
SMOVC C00274 BC00274 V=8.3  +MOVJ EC00274
SMOVL C00275 BC00275 V=8.3  +MOVJ EC00275
ARCOF
SFTOF3D
SMOVL C00276 BC00276 V=250.0  +MOVJ EC00276
SMOVL C00277 BC00277 V=250.0  +MOVJ EC00277
SFTON3D P043
SMOVL C00278 BC00278 V=166.7  +MOVJ EC00278
ARCON
SMOVC C00279 BC00279 V=8.3  +MOVJ EC00279
SMOVC C00280 BC00280 V=8.3  +MOVJ EC00280
SMOVC C00281 BC00281 V=8.3  +MOVJ EC00281
SMOVL C00282 BC00282 V=8.3  +MOVJ EC00282
ARCOF
SFTOF3D
SMOVL C00283 BC00283 V=166.7  +MOVJ EC00283
SMOVL C00284 BC00284 V=250.0  +MOVJ EC00284
MOVJ C00285 BC00285 VJ=30.00  +MOVJ EC00285 VJ=30.00
MACRO1 MJ#(0) ARGF9
MOVJ C00286 BC00286 VJ=15.00  +MOVJ EC00286 VJ=10.00
SFTON3D P044
SMOVL C00287 BC00287 V=166.7  +MOVJ EC00287
ARCON
SMOVL C00288 BC00288 V=9.2  +MOVJ EC00288
SMOVL C00289 BC00289 V=9.2  +MOVJ EC00289
ARCOF
SFTOF3D
SMOVL C00290 BC00290 V=250.0  +MOVJ EC00290
SFTON3D P045
SMOVL C00291 BC00291 V=166.7  +MOVJ EC00291
ARCON
SMOVL C00292 BC00292 V=9.2  +MOVJ EC00292
SMOVL C00293 BC00293 V=9.2  +MOVJ EC00293
SMOVL C00294 BC00294 V=9.2  +MOVJ EC00294
ARCOF
SMOVL C00295 BC00295 V=250.0  +MOVJ EC00295
SFTON3D P046
SMOVL C00296 BC00296 V=166.7  +MOVJ EC00296
ARCON
SMOVL C00297 BC00297 V=9.2  +MOVJ EC00297
SMOVL C00298 BC00298 V=9.2  +MOVJ EC00298
ARCOF
SFTOF3D
SMOVL C00299 BC00299 V=166.7  +MOVJ EC00299
SMOVL C00300 BC00300 V=250.0  +MOVJ EC00300
SMOVL C00301 BC00301 V=250.0  +MOVJ EC00301
SMOVL C00302 BC00302 V=250.0  +MOVJ EC00302
SFTON3D P045
SMOVL C00303 BC00303 V=166.7  +MOVJ EC00303
ARCON
SMOVL C00304 BC00304 V=10.0  +MOVJ EC00304
ARCOF
SMOVL C00305 BC00305 V=250.0  +MOVJ EC00305
SMOVL C00306 BC00306 V=333.3  +MOVJ EC00306
SFTON3D P044
SMOVL C00307 BC00307 V=166.7  +MOVJ EC00307
ARCON
SMOVL C00308 BC00308 V=10.0  +MOVJ EC00308
ARCOF
SMOVL C00309 BC00309 V=250.0  +MOVJ EC00309
MOVJ C00310 BC00310 VJ=20.00  +MOVJ EC00310 VJ=10.00
MOVJ C00311 BC00311 VJ=40.00  +MOVJ EC00311 VJ=10.00
MOVJ C00312 BC00312 VJ=20.00  +MOVJ EC00312 VJ=10.00
SFTON3D P050
SMOVL C00313 BC00313 V=166.7  +MOVJ EC00313
ARCON
SMOVL C00314 BC00314 V=9.2  +MOVJ EC00314
SMOVL C00315 BC00315 V=9.2  +MOVJ EC00315
ARCOF
SMOVL C00316 BC00316 V=166.7  +MOVJ EC00316
SFTON3D P049
SMOVL C00317 BC00317 V=166.7  +MOVJ EC00317
ARCON
SMOVL C00318 BC00318 V=9.2  +MOVJ EC00318
SMOVL C00319 BC00319 V=9.2  +MOVJ EC00319
SMOVL C00320 BC00320 V=9.2  +MOVJ EC00320
ARCOF
SMOVL C00321 BC00321 V=166.7  +MOVJ EC00321
SFTON3D P048
SMOVL C00322 BC00322 V=166.7  +MOVJ EC00322
ARCON
SMOVL C00323 BC00323 V=9.2  +MOVJ EC00323
SMOVL C00324 BC00324 V=9.2  +MOVJ EC00324
SMOVL C00325 BC00325 V=8.3  +MOVJ EC00325
ARCOF
SMOVL C00326 BC00326 V=166.7  +MOVJ EC00326
SMOVL C00327 BC00327 V=166.7  +MOVJ EC00327
SFTON3D P049
SMOVL C00328 BC00328 V=166.7  +MOVJ EC00328
ARCON
SMOVL C00329 BC00329 V=10.0  +MOVJ EC00329
ARCOF
SMOVL C00330 BC00330 V=250.0  +MOVJ EC00330
SFTON3D P050
SMOVL C00331 BC00331 V=200.0  +MOVJ EC00331
ARCON
SMOVL C00332 BC00332 V=10.0  +MOVJ EC00332
ARCOF
SFTOF3D
SMOVL C00333 BC00333 V=250.0  +MOVJ EC00333
MOVJ C00334 BC00334 VJ=60.00  +MOVJ EC00334 VJ=60.00
MOVJ C00335 BC00335 VJ=60.00  +MOVJ EC00335 VJ=60.00
MOVJ C00336 BC00336 VJ=100.00  +MOVJ EC00336 VJ=100.00
END
